TYPE ST_AxisVelBuf :
STRUCT
	SetVel  : ARRAY [0..999] OF LREAL;
	ActVel  : ARRAY [0..999] OF LREAL;
END_STRUCT
END_TYPE

(* stored: Version 1.1.0.1, ProductVersion 3.1.4024.9
   DUT ST_AxisVelBuf: Id {96910c6c-11e4-48a3-9590-9b0f6e771343} *)
